TYPE ST_TCCommands :
STRUCT
	arrTCCommands : ARRAY  [1..10] OF ST_Command;
		
END_STRUCT
END_TYPE

(* stored: Version 1.1.0.1, ProductVersion 3.1.4022.10
   DUT ST_TCCommands: Id {882879e8-7bd0-469e-887d-dba4a863692f} *)
